FUNCTION_BLOCK mqttCommsAdaptor IMPLEMENTS ITF_MachineDataService
VAR
	mqttComms : mqttCommunication;
END_VAR

METHOD SendStatus : INT
VAR_INPUT
	Status	: INT;
END_VAR
mqttComms.SendMQTTMessage(Status := TO_STRING(Status));
END_METHOD

END_FUNCTION_BLOCK

(* stored: Version 1.1.0.1, ProductVersion 3.1.4024.12
   POU mqttCommsAdaptor: Id {eb7e5bdd-a928-420d-8cb3-fc3345cd5725}, SpecialFunc None
   Method SendStatus: Id {4d0e1f9b-a446-45ae-baf6-8f00a2e8b9bd} *)
